FUNCTION_BLOCK Seq_1
VAR_INPUT
	// Basis-Inputs
	bExecute			:BOOL;				// Trigger für Ausführung von Sequenz
	iSysCommand			:eSystemCommand;	// Steuerungsvariabel von System (Resetten)
	iSysState			:eSystemState;		// Information über Zustand von System
	
	
	// Prozess-Inputs 
	Position_1			:sRoboterProzessVariablen;
	Position_DOWN		:sRoboterProzessVariablen;
	Position_UP			:sRoboterProzessVariablen;
	Position_2			:sRoboterProzessVariablen;
END_VAR
VAR_OUTPUT
	bDone				:BOOL;				// Information ob Sequenz ausgfeührt wurde
	bBusy				:BOOL;				// Information ob Sequenz im Moment ausgeführt wird
	bError				:BOOL;				// Information ob sich Sequenz in Fehlerzustand befindet
END_VAR
VAR
	// Sequenz-Zustände
	iState				:eSequenceState;
	
	// Startvariablen (FB soll nur bei einer steigenden Flanke gestartet werden)
	fTrigger			:R_TRIG;			// Erkennung einer steigenden Flanke für den Starte
	fSwitch				:SR;				// Setzen des Signals
	bSwitchResett		:BOOL;				// Resetten des Signals
	
	// Zustandsvariablen
	bStarten			:BOOL;
	bStoppen			:BOOL;
	bResetten			:BOOL;
	
	// Management-Variablen:
	bFinished			:BOOL;
	bInit				:BOOL;
	
	// Skill-Instanziierungen
	P2P_Bewegung		:Skill_Position_anfahren;
	Position			:sRoboterProzessVariablen;
	
END_VAR

// Aufrufen von Skills und Ablauf
Ablauf();	
Skills();

//_______________________________________________________________
// Reaktion auf Fehler
IF bError THEN
	iState := 3;
END_IF	

// Reaktion auf Input-Variablen: 
	// Starten
	fTrigger(CLK := bExecute);
	fSwitch(Set1 := fTrigger.Q);
	
	IF fSwitch.Q1 THEN
		bStarten := TRUE;
	ELSE
		bStarten := FALSE;
	END_IF
	
	// Stoppen
	IF iSysCommand = 3 THEN
		bStoppen := TRUE;	
	ELSE 
		bStoppen := FALSE;	
	END_IF
	
	// Stoppen
	IF iSysCommand = 4 THEN
		bResetten := TRUE;	
	ELSE 
		bResetten := FALSE;	
	END_IF



//_______________________________________________________________
// Zustandsmanagement
CASE iState OF 
	0:	// BEREIT
			// DO	
			fSwitch.RESET := FALSE;
				
			// TRANSITION
			IF bStarten THEN
				fSwitch.RESET := TRUE;
				iState := 1;																							// Starten des Objektes 
			END_IF
	// ________________________________________________________________________________			
	1:	// LAUFEND
			// DO
			bBusy := TRUE;	

			IF bStoppen THEN
				SFCReset := TRUE;
				bBusy := FALSE;
			END_IF	
			
			// TRANSITION
			IF bFinished THEN
				bFinished := FALSE;
				bBusy := FALSE;
				iState := 2;
			END_IF
			
			IF bInit THEN
				bInit := FALSE;
				SFCReset := FALSE;
				iState := 0;
			END_IF

	// ________________________________________________________________________________					
	2:	// ABGESCHLOSSEN
			// DO
			bDone := TRUE;			
						
			// TRANSITION
			IF bDone THEN
				bDone := FALSE;
				iState := 0;
			END_IF
	// ________________________________________________________________________________					
	3:	// FEHLER
			// DO
			bDone := FALSE;
			bBusy := FALSE;
			
			// TRANSITION
			IF bResetten THEN
				bError := FALSE;
				iState := 0;
			END_IF
			
END_CASE

ACTION Ablauf:
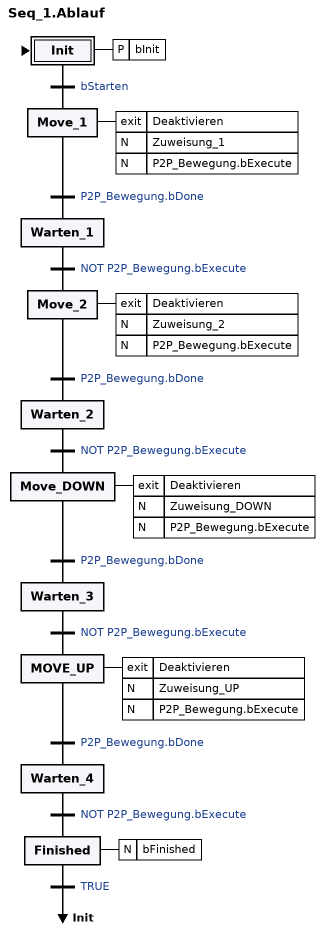
INITIAL_STEP Init:
    bInit(P);
END_STEP
TRANSITION FROM Init TO Move_1
    := bStarten;
END_TRANSITION
STEP Move_1:
    Deaktivieren(P0);  // exit action
    Zuweisung_1(N);
    P2P_Bewegung.bExecute(N);
END_STEP
TRANSITION FROM Move_1 TO Warten_1
    := P2P_Bewegung.bDone;
END_TRANSITION
STEP Warten_1:
END_STEP
TRANSITION FROM Warten_1 TO Move_2
    := NOT P2P_Bewegung.bExecute;
END_TRANSITION
STEP Move_2:
    Deaktivieren(P0);  // exit action
    Zuweisung_2(N);
    P2P_Bewegung.bExecute(N);
END_STEP
TRANSITION FROM Move_2 TO Warten_2
    := P2P_Bewegung.bDone;
END_TRANSITION
STEP Warten_2:
END_STEP
TRANSITION FROM Warten_2 TO Move_DOWN
    := NOT P2P_Bewegung.bExecute;
END_TRANSITION
STEP Move_DOWN:
    Deaktivieren(P0);  // exit action
    Zuweisung_DOWN(N);
    P2P_Bewegung.bExecute(N);
END_STEP
TRANSITION FROM Move_DOWN TO Warten_3
    := P2P_Bewegung.bDone;
END_TRANSITION
STEP Warten_3:
END_STEP
TRANSITION FROM Warten_3 TO MOVE_UP
    := NOT P2P_Bewegung.bExecute;
END_TRANSITION
STEP MOVE_UP:
    Deaktivieren(P0);  // exit action
    Zuweisung_UP(N);
    P2P_Bewegung.bExecute(N);
END_STEP
TRANSITION FROM MOVE_UP TO Warten_4
    := P2P_Bewegung.bDone;
END_TRANSITION
STEP Warten_4:
END_STEP
TRANSITION FROM Warten_4 TO Finished
    := NOT P2P_Bewegung.bExecute;
END_TRANSITION
STEP Finished:
    bFinished(N);
END_STEP
TRANSITION FROM Finished TO Init
    := TRUE;
END_TRANSITION
END_ACTION

ACTION Deaktivieren:
P2P_Bewegung.bExecute := FALSE;
END_ACTION

ACTION Skills:
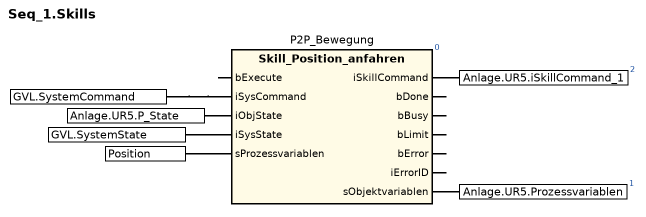
P2P_Bewegung(
    iSysCommand := GVL.SystemCommand,
    iObjState := Anlage.UR5.P_State,
    iSysState := GVL.SystemState,
    sProzessvariablen := Position); // Skill_Position_anfahren
Anlage.UR5.Prozessvariablen := P2P_Bewegung.sObjektvariablen;
Anlage.UR5.iSkillCommand_1 := P2P_Bewegung.iSkillCommand;
END_ACTION

ACTION Zuweisung_1:
Position := Position_1;
END_ACTION

ACTION Zuweisung_2:
Position := Position_2;
END_ACTION

ACTION Zuweisung_DOWN:
Position := Position_DOWN;
END_ACTION

ACTION Zuweisung_UP:
Position := Position_UP;
END_ACTION

END_FUNCTION_BLOCK

(* stored: Version 1.1.0.1
   POU Seq_1: Id {4e6711ea-ed1c-4254-8be6-d45b1ea5b2a6}, SpecialFunc None
   Folder 00_Hilfsaktionen: Id {9551f1fd-3283-49a9-864c-07abdc518f41}
   Folder 01_Zusweisung: Id {9e099ea1-4c50-4b6b-80e4-3448498f579a}
   Action Ablauf: Id {a51db42b-1e45-453f-ae91-17e0b4bf9c4f}
   Action Deaktivieren: Id {794dff7e-5fd1-43f4-b7d2-a9e5284cf510}
   Action Skills: Id {be3da68c-b614-492f-8b70-a1b7e3adc248}
   Action Zuweisung_1: Id {4f3116a9-3ff2-4b0c-8a6f-0b27a684be9a}
   Action Zuweisung_2: Id {64ea0b0e-bf22-49c7-bc8c-2f73002044aa}
   Action Zuweisung_DOWN: Id {53219e2a-818a-43c1-8682-428e3cb1d6f2}
   Action Zuweisung_UP: Id {9b099142-50b6-41b3-977a-da8325f4acd5} *)
